(*********************************** G.D S.p.A. - Technical Department ***********************************
============= PROGRAM INFO ============
FOLDER:             TBD
MACHINES INVOLVED:  TBD 

============= DESCRIPTION =============
csp machine declaration

============= REVISIONS ===============
Date		Version	 	Author      	Description             
----------	-------		------------  	--------------------------------------------
2019/04/05 	0000.00	 	M.Grasso		Creation of the PRG

**********************************************************************************************************)
(*$R process_ref := prc; $*)
PROGRAM csp_transfer_accumulator_finger
VAR
	
	prc:											process;
	prc_path:										STRING;
	
	cam_id: INT;
END_VAR

_read_var_input();

_object_manager();

IF NOT objects_running()
THEN
	RETURN;	
END_IF

_read_process_image();

_mode_manager();

_set_runtime_properties();

(********************************* BODY *********************************)
IF csp_main_brand.count = '48Count'
	THEN
		cam_id := 39;
ELSE 
	cam_id := 34;
END_IF
(************************************************************************)

_handle_messages();

_write_output();

ACTION _handle_messages:
;
END_ACTION

ACTION _handle_process_test:
;
END_ACTION

ACTION _mode_manager:
IF process_mode_req_is_pending(prc)
THEN
    process_apply_mode_req_first_step(prc);
    CASE process_get_mode(prc) OF
        MODE_TO_ABSENT:
			;
        MODE_TO_INACTIVE:
			;
        MODE_TO_TEST:
			;
        MODE_TO_OPERATIONAL:
			;
    END_CASE
    process_apply_mode_req_second_step(prc);
END_IF
END_ACTION

ACTION _object_manager:
IF objects_initialization()
THEN
	sub_process_init(
		object_name					:= 'csp_transfer_accumulator_finger.prc', 
		process						:= csp_transfer_accumulator.prc, 
		CONVERSION_this				:= prc);
		
	prc_path 						:= process_get_path(prc);
END_IF

IF objects_running()
THEN
	process_cycle(prc);
END_IF
END_ACTION

ACTION _read_process_image:
;
END_ACTION

ACTION _read_var_input:
;
END_ACTION

ACTION _set_runtime_properties:
;
END_ACTION

ACTION _write_output:
;
END_ACTION

END_PROGRAM

(* stored: Version 1.1.0.1, ProductVersion 3.1.4024.3
   POU csp_transfer_accumulator_finger: Id {a881e923-c709-4e7f-add5-2b1803f72602}, SpecialFunc None
   Action _handle_messages: Id {16c89b0d-f81c-45f8-9d60-9322c8a07ad2}
   Action _handle_process_test: Id {e00ef06c-acbb-4c6b-bf07-816a3e52f51e}
   Action _mode_manager: Id {6bac2fa9-e36c-4a21-a1c1-62f262d3a66c}
   Action _object_manager: Id {94a603e6-f99a-4901-81c0-48a80a1d5b69}
   Action _read_process_image: Id {5fcc2069-935b-4355-aab8-2b0a47286d0d}
   Action _read_var_input: Id {c11ea068-bed9-4cc4-8392-eab15c39ce7b}
   Action _set_runtime_properties: Id {13292848-b619-4a52-8b10-cc8b35a33180}
   Action _write_output: Id {dba8158e-61af-4e37-8115-c9a9ea73976f} *)
